// TwinCAT 3 PLC project _02_Tests
// ProgramVersion: 3.1.4026.18
// libraries:
//   Tc2_Standard, * (Beckhoff Automation GmbH)
//   Tc2_System, * (Beckhoff Automation GmbH)
//   StageCore, * (_)
//   StageUtils, * (_)
// project tree:
//   Broadcast/ TestCall.TcPOU, Test_Broadcast_FillAndCoalesce.TcPOU, Test_Broadcast_FillAndMove.TcPOU
//   / PlcTask.TcTTO
//   MAIN/ MAIN.TcPOU
//   Tags/ Test_Tags_WildcardCmp.TcPOU
// (motion and I/O tree: see PLC project _01_simple)
// real-time tasks:
//   TASK PlcTask: cycle T#10ms, priority 20, ADS port 350
//   TASK PlcTask1: cycle T#10ms, priority 21, ADS port 351

CONFIGURATION _02_Tests
    RESOURCE PLC ON TwinCAT3
        TASK PlcTask(INTERVAL := T#10ms, PRIORITY := 21);
        PROGRAM MAIN WITH PlcTask : MAIN;
    END_RESOURCE
END_CONFIGURATION

// ---- MAIN/MAIN.TcPOU
PROGRAM MAIN
VAR
	// Broadcast tests
	// Use only one Broadcast test at the time!
	{define broadcast_test '01'} 
	{IF hasvalue (broadcast_test, '01')}
		broadcast_test		: Test_Broadcast_FillAndCoalesce;
	{ELSE}
		broadcast_test		: Test_Broadcast_FillAndMove;
	{END_IF}
	
	// Tags tests
	tags_test_01			: Test_Tags_WildcardCmp;

	debugInfo				: DebugInfo;

END_VAR

Runtime();

END_PROGRAM

// ---- Broadcast/Test_Broadcast_FillAndCoalesce.TcPOU
// ASSUME Param.RECEIVER_CAP = 20
// Fills _Ec.comp table with first batch of signals
// Then fills _Broadcast.entry table with second batch of signals.
// Signal 1 entries need to be moved to the end, _Broadcast.iFirst is now Signal 2.
// Signal 2 entries expand towards the position 1.
// Signal 3 entries need to be moved to the end.

// Fill _Broadcast.entry with 3rd batch of signals forcing table to coalesce

// At the end the entity range should be number of compoennets plus header.
FUNCTION_BLOCK Test_Broadcast_FillAndCoalesce IMPLEMENTS I_Execute
VAR_INPUT
	bTest: BOOL := TRUE;
END_VAR
VAR_OUTPUT
(*
	Resulting _Broadcast.entry table:
	1. Signal[1] - Header
	2. batch01[1, 1]
	3. batch01[1, 2]
	4. batch02[1, 1]
	5. batch02[1, 2]
	6. Signal[2] - Header
	7. batch02[2, 2]
	8. batch02[2, 1]
	9. batch01[2, 1]
	10. batch01[2, 2]
	11. Signal[3] - Header
	12. batch01[3, 1]
	13. batch02[3, 2]
	14. batch02[3, 1]
	15. batch01[3, 2]
	16. CoalSignal - Header
	17. coalBatch[1]
	18. coalBatch[2]
	19. coalBatch[3]
	20. EMPTY
*)
END_VAR
VAR
	exe: Execute(THIS^);	
	call: TestCall;

	ett: EntityStart;
		signal: ARRAY[1..3] OF Signal; // 3 headers
		dfgSignal: Signal;
		
		batch01: ARRAY[1..3, 1..2] OF Receiver := [3((Callable := call)), 2((Callable := call))]; // 6 entries
		batch02: ARRAY[1..3, 1..2] OF Receiver := [3((Callable := call)), 2((Callable := call))];	// another 6 entries
		dfgBatch: ARRAY[1..4] OF Receiver := [4((Callable := call))];
	end: EntityEnd;
	i, j: UDINT;
END_VAR

METHOD Execute
VAR_INPUT
	nPhase: INT := 0;
END_VAR
IF bTest THEN
	FOR i := 1 TO 3 DO
		FOR j := 1 TO 2 DO
			signal[i].Pair(batch01[i, j]);
		END_FOR
	END_FOR

	FOR i := 1 TO 3 DO
		FOR j := 1 TO 2 DO
			signal[i].Pair(batch02[i, j]);
		END_FOR
	END_FOR
	
	FOR i := 1 TO 4 DO
		dfgSignal.Pair(dfgBatch[i]);
	END_FOR

	bTest := FALSE;
END_IF
END_METHOD

END_FUNCTION_BLOCK

// ---- Broadcast/TestCall.TcPOU
FUNCTION_BLOCK TestCall IMPLEMENTS I_Callable
VAR_INPUT
END_VAR
VAR_OUTPUT
END_VAR
VAR
	nUdint		: UDINT;
END_VAR

METHOD Call
VAR_INPUT
	iArg	: StageCore.I_Arg;
END_VAR
nUdint := nUdint + 1;
END_METHOD

END_FUNCTION_BLOCK

// ---- Broadcast/Test_Broadcast_FillAndMove.TcPOU
// ASSUME Param.RECEIVER_CAP = 20
// Fills _Ec.comp table with first batch of signals
// Then fills _Broadcast.entry table with second batch of signals.
// Signal 1 entries need to be moved to the end, _Broadcast.iFirst is now Signal 2.
// Signal 2 entries expand towards the position 1.
// Signal 3 entries need to be moved to the end.
// At the end the entity range should be number of compoennets plus header.
FUNCTION_BLOCK Test_Broadcast_FillAndMove IMPLEMENTS I_Execute
VAR_INPUT
	bTest		: BOOL := TRUE;
END_VAR
VAR_OUTPUT
(*
	Resulting _Broadcast.entry table:
	1. EMPTY
	2. Signal[2] - Header
	3. batch02[2, 2]
	4. batch02[2, 1]
	5. batch01[2, 1]
	6. batch01[2, 2]
	7. EMPTY
	8. EMPTY
	9. EMPTY
	10. Signal[1] - Header
	11. batch01[1, 1]
	12. batch01[1, 2]
	13. batch02[1, 1]
	14. batch02[1, 2]
	15. Signal[3] - Header
	16. batch01[3, 1]
	17. batch01[3, 2]
	18. batch02[3, 1]
	19. batch02[3, 2]
	20. EMPTY
*)
END_VAR
VAR
	exe					: Execute(THIS^);	
	call				: TestCall;
	
	ett					: EntityStart;
		signal				: ARRAY[1..3] OF Signal; // 3 headers
		
		batch01				: ARRAY[1..3, 1..2] OF Receiver := [3((Callable := call)), 2((Callable := call))]; // 6 entries
		batch02				: ARRAY[1..3, 1..2] OF Receiver := [3((Callable := call)), 2((Callable := call))];	// another 6 entries
	end					: EntityEnd;
	i, j				: UDINT;
END_VAR

METHOD Execute
VAR_INPUT
	nPhase: INT := 0;
END_VAR
IF bTest THEN
	FOR i := 1 TO 3 DO
		FOR j := 1 TO 2 DO
			signal[i].Pair(batch01[i, j]);
		END_FOR
	END_FOR

	FOR i := 1 TO 3 DO
		FOR j := 1 TO 2 DO
			signal[i].Pair(batch02[i, j]);
		END_FOR
	END_FOR

	bTest := FALSE;
END_IF
END_METHOD

END_FUNCTION_BLOCK

// ---- Tags/Test_Tags_WildcardCmp.TcPOU
FUNCTION_BLOCK Test_Tags_WildcardCmp IMPLEMENTS I_Execute
VAR_INPUT
	bTest			: BOOL := TRUE;
END_VAR
VAR_OUTPUT
	nMatchResult	: USINT;
END_VAR
VAR
	exe				: Execute(THIS^);
	sAddress		: Str := 'abc.def.ghi.jkl';
	sPattern		: ARRAY[1..10] OF Str := ['abc.def.ghi.jkl', 'abc.*', '*.ghi.*', '*.ghi', '*.jkl.*', 'abc.*.*.jkl', 'abc.*.*.*', 'abc.def.xyz.jkl', 'abc.def', '*'];
	nResult			: ARRAY[1..10] OF Result;
	nExpected		: ARRAY[1..10] OF Result := [Ok, Ok, Ok, Err.NoMatch, Ok, Ok, Ok, Err.NoMatch, Err.NoMatch, Ok];
	i				: USINT;
END_VAR

METHOD Execute
VAR_INPUT
	nPhase: INT := 0;
END_VAR
IF bTest THEN
	FOR i := 1 TO 10 DO
		nResult[i] := MatchPath(sAddress, sPattern[i]);
		IF nResult[i] = nExpected[i] THEN
			nMatchResult := nMatchResult + 1;
		END_IF
	END_FOR
	
	bTest := FALSE;
END_IF
END_METHOD

END_FUNCTION_BLOCK
